// TwinCAT 3 PLC project PlcAdsCounter
// ProgramVersion: 3.1.4023.0
// libraries:
//   Tc2_Standard, * (Beckhoff Automation GmbH)
//   Tc2_System, * (Beckhoff Automation GmbH)
//   Tc3_Module, * (Beckhoff Automation GmbH)
// project tree:
//   / PlcTask.TcTTO
//   POUs/ MAIN.TcPOU
// real-time tasks:
//   TASK TaskMain: cycle T#10ms, priority 1, ADS port 350
//   TASK PlcTask: cycle T#10ms, priority 20, ADS port 351
// variable links:
//   PlcAdsCounter/PlcAdsCounter Instance <-> beispiele/beispiele_Obj6 (ModuleBeispiel4PlcIoAdsCommunication)
//     PlcTask Outputs/MAIN.x <-> Inputs/PLCX
//   beispiele/beispiele_Obj2 (ModuleBeispiel2Out) <-> beispiele/beispiele_Obj3 (ModuleBeispiel2In)
//     Outputs/Fancy <-> Inputs/Fancy

CONFIGURATION PlcAdsCounter
    RESOURCE PLC ON TwinCAT3
        TASK PlcTask(INTERVAL := T#10ms, PRIORITY := 20);
        PROGRAM MAIN WITH PlcTask : MAIN;
    END_RESOURCE
END_CONFIGURATION

// ---- POUs/MAIN.TcPOU
PROGRAM MAIN
VAR
	fbCounter: TON;
	tCount: TIME := T#1S;
	up: BOOL := TRUE;
	x AT %QB1: USINT := 0;
	doCount: BOOL := TRUE;
END_VAR

// Einfaches Programm, welches von 0 bis 5 hoch und wieder hinunter zählt

// Jede Sekunde Wert inkrementieren / dekrementieren
fbCounter(IN := TRUE, PT := tCount, Q => doCount);
IF doCount THEN
	IF up THEN
		x := x + 1;
	ELSE
		x := x - 1;
	END_IF;
	
	// Zählrichtung evaluieren 
	IF x = 5 THEN
		up := FALSE;
	ELSIF x = 0 THEN
		up := TRUE;
	END_IF

	doCount := FALSE;
	fbCounter(IN := FALSE);
END_IF

END_PROGRAM
